// TIA Portal V19 export
TYPE "Positioning_DOL_Machine_Config"
// stored: Access Published
   STRUCT
      DelayMissingCondition : Time := T#3s;
      CyclicOBTime_ms : LReal := 10.0;
      Ax : "OOAx_Config";
      Ax_UM2 : "udt_LinTranformation";
      S120 : Struct
         SpeedMotor : "SpeedMotor_Config";
         PowerOffDelay : Time := T#1500ms;
         StandstillVelocity : LReal;
         AccTime : LReal;   // [s]
         DecTime : LReal;   // [s]
      END_STRUCT;
      Fan : Struct
         Presence : Bool := FALSE;
         DelayOff : Time := T#10m;
      END_STRUCT;
      Brake_Presence : Bool := FALSE;
   END_STRUCT;
   // Ax_UM2."m" := 1.0;
   // Ax_UM2.q := 0.0;
   // S120.SpeedMotor.ReferenceVelocity := 2000.0;
   // S120.SpeedMotor.InvertDirection := FALSE;
END_TYPE
